// TIA Portal V20 export
DATA_BLOCK "LBP_ReadVar_DB_R_Param"   // DB129
// stored: InstanceOfName LBP_ReadVar, InstanceOfType FB
"LBP_ReadVar"
   // VAR_INPUT
   //    Req : Bool;
   //    NumVar : Int;
   //    Addr1 : Variant;
   //    Unit1 : Byte;
   //    Column1 : Word;
   //    Line1 : Word;
   //    Addr2 : Variant;
   //    Unit2 : Byte;
   //    Column2 : Word;
   //    Line2 : Word;
   //    Addr3 : Variant;
   //    Unit3 : Byte;
   //    Column3 : Word;
   //    Line3 : Word;
   //    Addr4 : Variant;
   //    Unit4 : Byte;
   //    Column4 : Word;
   //    Line4 : Word;
   //    Addr5 : Variant;
   //    Unit5 : Byte;
   //    Column5 : Word;
   //    Line5 : Word;
   //    Addr6 : Variant;
   //    Unit6 : Byte;
   //    Column6 : Word;
   //    Line6 : Word;
   //    Addr7 : Variant;
   //    Unit7 : Byte;
   //    Column7 : Word;
   //    Line7 : Word;
   //    Addr8 : Variant;
   //    Unit8 : Byte;
   //    Column8 : Word;
   //    Line8 : Word;
   // END_VAR
   // VAR_OUTPUT
   //    Error : Bool;
   //    NDR : Bool;
   //    State : Word;
   // END_VAR
   // VAR_IN_OUT
   //    RD1 : Variant;
   //    RD2 : Variant;
   //    RD3 : Variant;
   //    RD4 : Variant;
   //    RD5 : Variant;
   //    RD6 : Variant;
   //    RD7 : Variant;
   //    RD8 : Variant;
   // END_VAR
   // VAR
   //    ident : Byte;
   //    regist : Bool;
   //    flanke : Bool;
   //    progtest : Bool;
   //    err_cls_cod : Word;
   //    err_stat : Word;
   //    s_fifoRef : UInt;
   //    s_Reserved1 : Word;
   //    s_Reserved2 : DWord;
   //    s_Reserved3 : DWord;
   // END_VAR
BEGIN
END_DATA_BLOCK
